// TIA Portal V21 export
VAR_GLOBAL   // PLC tag table "GruppoRiempiReciveAnalogici"
END_VAR
VAR_GLOBAL CONSTANT   // user constants
   K_SegnaleDaGruppoRiempi_Temperatura : Int := 1;
END_VAR
